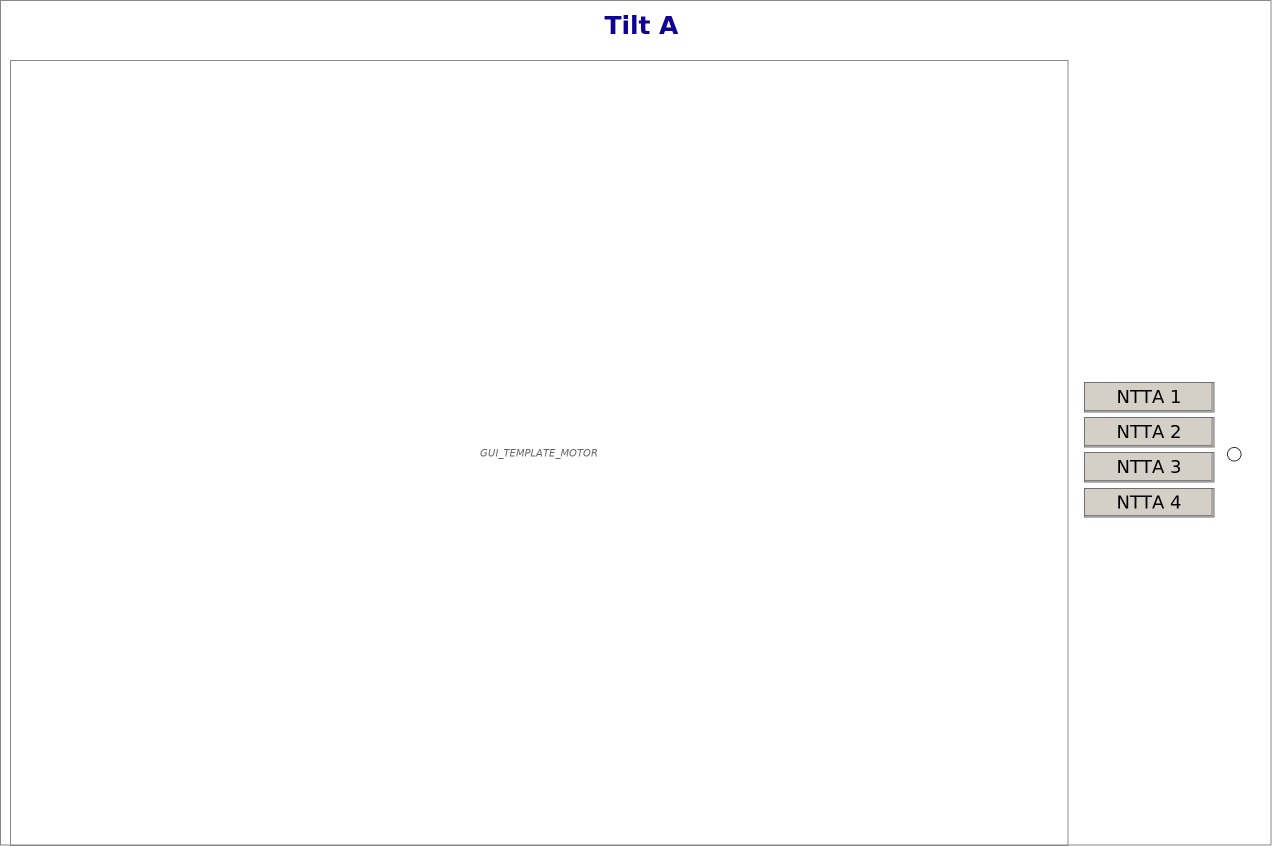
VISUALIZATION VISU_HMI_TILT_A  // 1272x846
    Group (10,60 1262x786)
        Frame (0,0 1058x786)
            shows GUI_TEMPLATE_MOTOR(m_Instance := MAIN.nott_ics.TipTilt.ptrTiltActuatorsA[MAIN.nott_ics.TipTilt.guiTiltActuatorsAIndex]^)
        Group (1074,322 188x142)
            RadioButton (141,2 47x140), variable: MAIN.nott_ics.TipTilt.guiTiltActuatorsAIndex-1
                Areas[0]: Text=Radiobutton
                Areas[1]: Text=Radiobutton
            Button (0,0 130x30), "NTTA 1"
                OnMouseClick: execute { MAIN.nott_ics.TipTilt.guiTiltActuatorsAIndex := 1; }
            Button (0,35 130x30), "NTTA 2"
                OnMouseClick: execute { MAIN.nott_ics.TipTilt.guiTiltActuatorsAIndex := 2; }
            Button (0,70 130x30), "NTTA 3"
                OnMouseClick: execute { MAIN.nott_ics.TipTilt.guiTiltActuatorsAIndex := 3; }
            Button (0,106 130x29), "NTTA 4"
                OnMouseClick: execute { MAIN.nott_ics.TipTilt.guiTiltActuatorsAIndex := 4; }
    Label (542,10 199x30), "Tilt A"
END_VISUALIZATION

(* stored: Version 1.1.0.1, ProductVersion 3.1.4024.14
   Visu VISU_HMI_TILT_A: Id {252baf16-c431-4a95-b610-76b6bfb52b48} *)
